FUNCTION_BLOCK FB_Motion
VAR_INPUT
	bStart: BOOL;
	nPosition: LREAL;
	bStopEx: BOOL;
	bMoveAbs: BOOL;
END_VAR
VAR_OUTPUT
	bBusy: BOOL;
	bDone: BOOL;
	bStopDone: BOOL;
END_VAR
VAR
	MC_Power1: MC_Power;
	MC_MoveAbsolute1: MC_MoveAbsolute;
	MC_Stop1: MC_Stop;

END_VAR

MC_Power1(
	Axis:=Axis1 , 
	Enable:=TRUE , 
	Enable_Positive:=TRUE , 
	Enable_Negative:=TRUE , 
	Override:=100, 
	BufferMode:= , 
	Options:= , 
	Status=> , 
	Busy=> , 
	Active=> , 
	Error=> , 
	ErrorID=> );
	
	
	MC_MoveAbsolute1(
	Axis:= Axis1, 
	Execute:=bMoveAbs , 
	Position:=nPosition , 
	Velocity:= 8000, 
	Acceleration:= , 
	Deceleration:= , 
	Jerk:= , 
	BufferMode:= , 
	Options:= , 
	Done=>bDone , 
	Busy=>bBusy , 
	Active=> , 
	CommandAborted=> , 
	Error=> , 
	ErrorID=> );
	
			MC_Stop1(
	Axis:=Axis1 , 
	Execute:=bStopEx , 
	Deceleration:= , 
	Jerk:= , 
	Options:= , 
	Done=>bStopDone , 
	Busy=> , 
	Active=> , 
	CommandAborted=> , 
	Error=> , 
	ErrorID=> );

END_FUNCTION_BLOCK

(* stored: Version 1.1.0.1, ProductVersion 3.1.4022.16
   POU FB_Motion: Id {86bc4b4a-a009-4992-926e-1ac1c48eab02}, SpecialFunc None *)
